
FUNCTION CB_dword_to_word : WORD

TITLE = ' Convert a double word into an word '
VERSION : '1.0'
AUTHOR  : CB
NAME    : DintToWo
FAMILY  : TNI

VAR_INPUT
    IN : DWORD;
END_VAR

VAR_TEMP

END_VAR

BEGIN

CB_dword_to_word := DWORD_TO_WORD(IN);

END_FUNCTION
